// TIA Portal V18 export
// export: Created 2026-06-08T17:01:58.3891487Z, ExportSetting WithDefaults, DisplayName Totally Integrated Automation Portal, DisplayVersion V18, DisplayName TIA Portal Openness, DisplayVersion V18, DisplayName TIA Portal Version Control Interface, DisplayVersion V18, DisplayName STEP 7 Professional, DisplayVersion V18, DisplayName STEP 7 Safety, DisplayVersion V18, DisplayName WinCC Professional, DisplayVersion V18
FUNCTION "M1_I/O" : Void   // FC4, LAD
{ S7_Optimized_Access := 'TRUE' }
VERSION : 0.1
// stored: AutoNumber true, IsIECCheckEnabled false, SetENOAutomatically false, UDAEnableTagReadback false
BEGIN

REGION Network 1
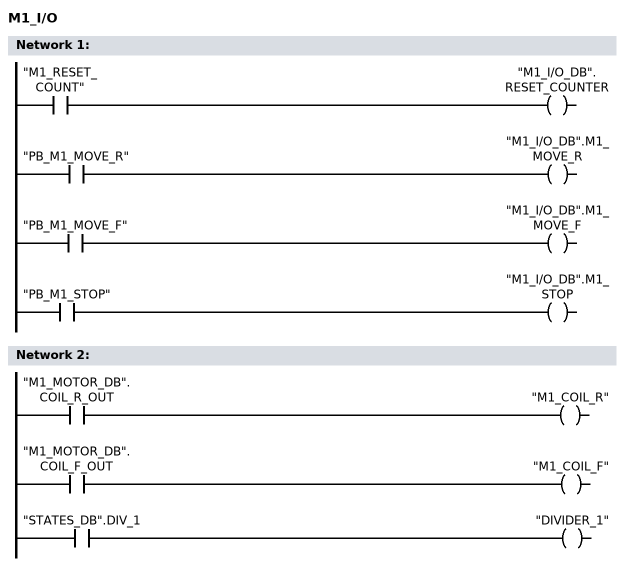
   RUNG wire#powerrail
      Contact( "M1_RESET_COUNT" )
      Coil( "M1_I/O_DB".RESET_COUNTER )
   END_RUNG
   RUNG wire#powerrail
      Contact( "PB_M1_MOVE_R" )
      Coil( "M1_I/O_DB".M1_MOVE_R )
   END_RUNG
   RUNG wire#powerrail
      Contact( "PB_M1_MOVE_F" )
      Coil( "M1_I/O_DB".M1_MOVE_F )
   END_RUNG
   RUNG wire#powerrail
      Contact( "PB_M1_STOP" )
      Coil( "M1_I/O_DB".M1_STOP )
   END_RUNG
   // the same network as SCL:
   "M1_I/O_DB".RESET_COUNTER := "M1_RESET_COUNT";
   "M1_I/O_DB".M1_MOVE_R := "PB_M1_MOVE_R";
   "M1_I/O_DB".M1_MOVE_F := "PB_M1_MOVE_F";
   "M1_I/O_DB".M1_STOP := "PB_M1_STOP";
END_REGION

REGION Network 2
   RUNG wire#powerrail
      Contact( "M1_MOTOR_DB".COIL_R_OUT )
      Coil( "M1_COIL_R" )
   END_RUNG
   RUNG wire#powerrail
      Contact( "M1_MOTOR_DB".COIL_F_OUT )
      Coil( "M1_COIL_F" )
   END_RUNG
   RUNG wire#powerrail
      Contact( "STATES_DB".DIV_1 )
      Coil( "DIVIDER_1" )
   END_RUNG
   // the same network as SCL:
   "M1_COIL_R" := "M1_MOTOR_DB".COIL_R_OUT;
   "M1_COIL_F" := "M1_MOTOR_DB".COIL_F_OUT;
   "DIVIDER_1" := "STATES_DB".DIV_1;
END_REGION
END_FUNCTION
